SUBAPPLICATION Uebung_004b4c_sub_AX (* Sub-Applikation für ein verriegelbares Toggle-Flip-Flop mit AE2-Adapter *)
  (* Standard: 61499-2; Description: Copyright (c) 2023 Meisterschulen am Ostbahnhof This program and the accompanying materials are made available under the terms of the Eclipse Public License 2.0 which is available at https://www.eclipse.org/legal/epl-2.0/ SPDX-License-Identifier: EPL-2.0 *)
  (* Version 1.0, 2026-04-19, Franz Höpfinger, Meisterschulen am Ostbahnhof, initial API and implementation and/or initial documentation *)
  PACKAGE Uebungen;
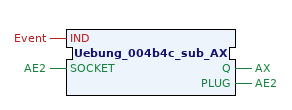
  EVENT_INPUT
    IND;
  END_EVENT
  SOCKETS
    SOCKET : adapter::types::bidirectional::AE2;
  END_SOCKETS
  PLUGS
    Q : adapter::types::unidirectional::AX;
    PLUG : adapter::types::bidirectional::AE2;
  END_PLUGS
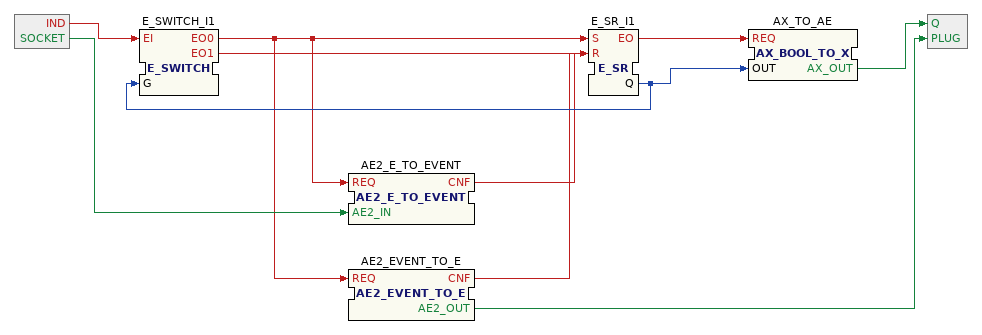
  FBS
    E_SR_I1 : iec61499::events::E_SR;
    E_SWITCH_I1 : iec61499::events::E_SWITCH;
    AE2_EVENT_TO_E : adapter::conversion::bidirectional::AE2_EVENT_TO_E;
    AE2_E_TO_EVENT : adapter::conversion::bidirectional::AE2_E_TO_EVENT;
    AX_TO_AE : adapter::conversion::unidirectional::AX_BOOL_TO_X;
  END_FBS
  EVENT_CONNECTIONS
    E_SWITCH_I1.EO0 TO E_SR_I1.S;
    E_SWITCH_I1.EO1 TO E_SR_I1.R;
    IND TO E_SWITCH_I1.EI;
    E_SWITCH_I1.EO0 TO AE2_EVENT_TO_E.REQ;
    AE2_E_TO_EVENT.CNF TO E_SR_I1.R;
    AE2_EVENT_TO_E.CNF TO E_SR_I1.R;
    E_SWITCH_I1.EO0 TO AE2_E_TO_EVENT.REQ;
    E_SR_I1.EO TO AX_TO_AE.REQ;
  END_CONNECTIONS
  DATA_CONNECTIONS
    E_SR_I1.Q TO E_SWITCH_I1.G;
    E_SR_I1.Q TO AX_TO_AE.OUT;
  END_CONNECTIONS
  ADAPTER_CONNECTIONS
    SOCKET TO AE2_E_TO_EVENT.AE2_IN;
    AE2_EVENT_TO_E.AE2_OUT TO PLUG;
    AX_TO_AE.AX_OUT TO Q;
  END_CONNECTIONS
END_SUBAPPLICATION
